(* CODESYS project ast_v1_0.library
   Company: Deprag
   Version: 1.0
   Placeholder: AST_V1_0
   Title: AST_V1_0

Project tree, tasks and I/O mapping:
  Data types/
    AST11/
      data type tAST11
      data type tAST11control
      data type tAST11data
      data type tAST11Rx
      data type tAST11state
      data type tAST11Tx
    AST40/
      data type tAST40
      data type tAST40control
      data type tAST40data
      data type tAST40Rx
      data type tAST40state
      data type tAST40Tx
    AST6/
      data type tAST6
      data type tAST6control
      data type tAST6data
      data type tAST6Rx
      data type tAST6state
      data type tAST6Tx
  Global Variables/
    global variables Globale_Variablen
  POUs/
    AST11/
      function block FB_AST11 [ST]: mthConvertControlSignal, mthConvertFinalData, mthConvertStatusSignal
      function FC_ConvertUnitAST11 [ST]
    AST40/
      function block FB_AST40 [ST]: mthConvertControlSignal, mthConvertFinalData, mthConvertStatusSignal
      function FC_ConvertUnitAST40 [ST]
    AST6/
      function block FB_AST6 [ST]: mthConvertControlSignal, mthConvertFinalData, mthConvertStatusSignal
      function FC_ConvertUnitAST6 [ST]
    Internal/
      function Merge_Byte2DInt [ST]
      function Merge_Byte2Int [ST]
      function Merge_Byte2Real [ST]
      function Split_Int2Byte [ST]
  Version/
    global variables Global_Version
  Visualizations/
*)

// Data types/AST11/tAST11
TYPE tAST11 :
	STRUCT
		Control			: tAST11control;
		State			: tAST11state;
		Data			: tAST11data;
	END_STRUCT
END_TYPE

// Data types/AST11/tAST11control
TYPE tAST11control :
	STRUCT
		Start			: BOOL := FALSE;
		Stop			: BOOL := FALSE;
		AutoStop		: BOOL := FALSE;
		Reload			: BOOL := FALSE;
		StartRelease	: BOOL := FALSE;
		ProgIn2			: BOOL := FALSE;
		FC_PartSensor	: BOOL := FALSE;
		FC_ReleasePart	: BOOL := FALSE;
		FC_ErrorReset	: BOOL := FALSE;
		DataSaved		: BOOL := FALSE;
		ResetPowerunit	: BOOL := FALSE;
		ResetMaintenance: BOOL := FALSE;
		ResetCycleStarted: BOOL := FALSE;
		Heartbeat		: BOOL := FALSE;
		ProgramNo		: INT := 0;
	END_STRUCT
END_TYPE

// Data types/AST11/tAST11data
TYPE tAST11data :
	STRUCT
		fdProg			: INT;
		fdStatus		: INT;
		fdTime			: REAL;

		fdStep1			: DINT;
		fdTorque1		: REAL;
		fdAngle1		: DINT;

		fdStep2			: DINT;
		fdTorque2		: REAL;
		fdAngle2		: DINT;

		fdStep3			: DINT;
		fdTorque3		: REAL;
		fdAngle3		: DINT;

		fdStepNOk		: DINT;
		fdTorqueNOk		: REAL;
		fdAngleNOk		: DINT;

		fdTorqueUnit	: INT;

		FC_Status		: INT;
		FC_TargetCount	: INT;
		FC_ActualCount	: INT;
	END_STRUCT
END_TYPE

// Data types/AST11/tAST11Rx
TYPE
	tAST11Rx : ARRAY[0..71] OF BYTE;
END_TYPE

// Data types/AST11/tAST11state
TYPE tAST11state :

	STRUCT
		SystemOK		: BOOL := FALSE;
		Ready			: BOOL := FALSE;
		OK				: BOOL := FALSE;
		NOK				: BOOL := FALSE;
		FC_PartActive	: BOOL := FALSE;
		FC_ChangePart	: BOOL := FALSE;
		ProgOut8		: BOOL := FALSE;
		DataAvailable	: BOOL := FALSE;

		ExtStop			: BOOL := FALSE;
		CycleActive		: BOOL := FALSE;
		CycleStarted	: BOOL := FALSE;
		Heartbeat		: BOOL := FALSE;

		SysStatus		: INT := 0;
	END_STRUCT
END_TYPE

// Data types/AST11/tAST11Tx
TYPE tAST11Tx : ARRAY[0..3] OF BYTE;
END_TYPE

// Data types/AST40/tAST40
TYPE tAST40 :
	STRUCT
		Control			: tAST40control;
		State			: tAST40state;
		Data			: tAST40data;
	END_STRUCT
END_TYPE

// Data types/AST40/tAST40control
TYPE tAST40control :
	STRUCT
		FCErrReset		: BOOL := FALSE;
		FCPartSensor	: BOOL := FALSE;
		FCReleasePart	: BOOL := FALSE;
		ReleaseStart	: BOOL := FALSE;
		Start			: BOOL := FALSE;
		Reload			: BOOL := FALSE;
		In1				: BOOL := FALSE;
		In2				: BOOL := FALSE;
		In3				: BOOL := FALSE;
		In4				: BOOL := FALSE;
		Res1			: BOOL := FALSE;
		Res2			: BOOL := FALSE;
		Res3			: BOOL := FALSE;
		Res4			: BOOL := FALSE;
		Res5			: BOOL := FALSE;
		Res6			: BOOL := FALSE;
		ProgramNo		: INT  := 0;
		In5				: BOOL := FALSE;
		In6				: BOOL := FALSE;
		In7				: BOOL := FALSE;
		In8				: BOOL := FALSE;
		In9				: BOOL := FALSE;
		In10			: BOOL := FALSE;
		In11			: BOOL := FALSE;
		In12			: BOOL := FALSE;
		UniInRes1		: BOOL := FALSE;
		UniInRes2		: BOOL := FALSE;
		UniInRes3		: BOOL := FALSE;
		UniInRes4		: BOOL := FALSE;
		UniInRes5		: BOOL := FALSE;
		UniInRes6		: BOOL := FALSE;
		UniInRes7		: BOOL := FALSE;
		UniInRes8		: BOOL := FALSE;
		DataSaved		: BOOL := FALSE;
		Heartbeat		: BOOL := FALSE;
		InRes1			: BOOL := FALSE;
		InRes2			: BOOL := FALSE;
		InRes3			: BOOL := FALSE;
		InRes4			: BOOL := FALSE;
		InRes5			: BOOL := FALSE;
		InRes6			: BOOL := FALSE;
		InRes7			: BOOL := FALSE;
		InRes8			: BOOL := FALSE;
		InRes9			: BOOL := FALSE;
		InRes10			: BOOL := FALSE;
		InRes11			: BOOL := FALSE;
		InRes12			: BOOL := FALSE;
		InRes13			: BOOL := FALSE;
		InRes14			: BOOL := FALSE;
	END_STRUCT
END_TYPE

// Data types/AST40/tAST40data
TYPE tAST40data :
	STRUCT
		fdProg			: INT;
		fdStatus		: INT;
		fdTime			: REAL;

		fdStep1			: DINT;
		fdMinTorque1	: REAL;
		fdTarTorque1	: REAL;
		fdMaxTorque1	: REAL;
		fdTorque1		: REAL;
		fdMinAngle1		: DINT;
		fdTarAngle1		: DINT;
		fdMaxAngle1		: DINT;
		fdAngle1		: REAL;

		fdStep2			: DINT;
		fdMinTorque2	: REAL;
		fdTarTorque2	: REAL;
		fdMaxTorque2	: REAL;
		fdTorque2		: REAL;
		fdMinAngle2		: DINT;
		fdTarAngle2		: DINT;
		fdMaxAngle2		: DINT;
		fdAngle2		: REAL;

		fdStep3			: DINT;
		fdMinTorque3	: REAL;
		fdTarTorque3	: REAL;
		fdMaxTorque3	: REAL;
		fdTorque3		: REAL;
		fdMinAngle3		: DINT;
		fdTarAngle3		: DINT;
		fdMaxAngle3		: DINT;
		fdAngle3		: REAL;

		fdStepNOk		: DINT;
		fdMinTorqueNOk	: REAL;
		fdTarTorqueNOk	: REAL;
		fdMaxTorqueNOk	: REAL;
		fdTorqueNOk		: REAL;
		fdMinAngleNOk	: DINT;
		fdTarAngleNOk	: DINT;
		fdMaxAngleNOk	: DINT;
		fdAngleNOk		: REAL;

		fdTorqueUnit	: INT;
	END_STRUCT
END_TYPE

// Data types/AST40/tAST40Rx
TYPE
	tAST40Rx : ARRAY[0..169] OF BYTE;
END_TYPE

// Data types/AST40/tAST40state
TYPE tAST40state :
	STRUCT
		SystemOK		: BOOL := FALSE;
		Ready			: BOOL := FALSE;
		OK				: BOOL := FALSE;
		NOK				: BOOL := FALSE;
		StatusHSres		: BOOL := FALSE;
		Sto1active		: BOOL := FALSE;
		Sto2active		: BOOL := FALSE;
		CycleActive		: BOOL := FALSE;
		ProgOut1		: BOOL := FALSE;
		ProgOut2		: BOOL := FALSE;
		ProgOut3		: BOOL := FALSE;
		ProgOut4		: BOOL := FALSE;
		FC_LockPart		: BOOL := FALSE;
		StatLTres		: BOOL := FALSE;
		FC_CycleDone	: BOOL := FALSE;
		Reload			: BOOL := FALSE;
		ProgOut5		: BOOL := FALSE;
		ProgOut6		: BOOL := FALSE;
		ProgOut7		: BOOL := FALSE;
		ProgOut8		: BOOL := FALSE;
		ProgOut9		: BOOL := FALSE;
		ProgOut10		: BOOL := FALSE;
		ProgOut11		: BOOL := FALSE;
		ProgOut12		: BOOL := FALSE;
		UniOutRes1		: BOOL := FALSE;
		UniOutRes2		: BOOL := FALSE;
		UniOutRes3		: BOOL := FALSE;
		UniOutRes4		: BOOL := FALSE;
		UniOutRes5		: BOOL := FALSE;
		UniOutRes6		: BOOL := FALSE;
		UniOutRes7		: BOOL := FALSE;
		UniOutRes8		: BOOL := FALSE;
		DataAvailable	: BOOL := FALSE;
		Heartbeat		: BOOL := FALSE;
		OutRes1			: BOOL := FALSE;
		OutRes2			: BOOL := FALSE;
		OutRes3			: BOOL := FALSE;
		OutRes4			: BOOL := FALSE;
		OutRes5			: BOOL := FALSE;
		OutRes6			: BOOL := FALSE;
		OutRes7			: BOOL := FALSE;
		OutRes8			: BOOL := FALSE;
		OutRes9			: BOOL := FALSE;
		OutRes10		: BOOL := FALSE;
		OutRes11		: BOOL := FALSE;
		OutRes12		: BOOL := FALSE;
		OutRes13		: BOOL := FALSE;
		OutRes14		: BOOL := FALSE;
		HW_FCErrReset	: BOOL := FALSE;
		HW_FCPartSensor	: BOOL := FALSE;
		HW_FCPartRelease: BOOL := FALSE;
		HW_ReleaseStart	: BOOL := FALSE;
		HW_Start		: BOOL := FALSE;
		HW_Reload		: BOOL := FALSE;
		HW_ProgIn1		: BOOL := FALSE;
		HW_ProgIn2		: BOOL := FALSE;
		HW_ProgIn3		: BOOL := FALSE;
		HW_ProgIn4		: BOOL := FALSE;
		HW_Res1			: BOOL := FALSE;
		HW_Res2			: BOOL := FALSE;
		HW_Res3			: BOOL := FALSE;
		HW_Res4			: BOOL := FALSE;
		HW_Res5			: BOOL := FALSE;
		HW_Res6			: BOOL := FALSE;
		AnalogStop		: INT  := 0;
		SysStatus		: INT  := 0;
	END_STRUCT
END_TYPE

// Data types/AST40/tAST40Tx
TYPE tAST40Tx : ARRAY[0..17] OF BYTE;
END_TYPE

// Data types/AST6/tAST6
TYPE tAST6 :
	STRUCT
		Control			: tAST6control;
		State			: tAST6state;
		Data			: tAST6data;
	END_STRUCT
END_TYPE

// Data types/AST6/tAST6control
TYPE tAST6control :
	STRUCT
		Start			: BOOL := FALSE;
		ProgIn1			: BOOL := FALSE;
		ProgIn2			: BOOL := FALSE;
		ProgIn3			: BOOL := FALSE;
		ProgIn4			: BOOL := FALSE;
		ProgIn5			: BOOL := FALSE;
		ProgIn6			: BOOL := FALSE;
		ProgramNo		: INT := 0;
		DataSaved		: BOOL := FALSE;
		Heartbeat		: BOOL := FALSE;
	END_STRUCT
END_TYPE

// Data types/AST6/tAST6data
TYPE tAST6data :
	STRUCT
		fdProg			: INT;
		fdStatus		: INT;
		fdTime			: REAL;

		fdStep1			: DINT;
		fdTorque1		: REAL;
		fdAngle1		: DINT;

		fdStep2			: DINT;
		fdTorque2		: REAL;
		fdAngle2		: DINT;

		fdStep3			: DINT;
		fdTorque3		: REAL;
		fdAngle3		: DINT;

		fdStepNOk		: DINT;
		fdTorqueNOk		: REAL;
		fdAngleNOk		: DINT;

		fdTorqueUnit	: INT;

	END_STRUCT
END_TYPE

// Data types/AST6/tAST6Rx
TYPE
	tAST6Rx : ARRAY[0..169] OF BYTE;
END_TYPE

// Data types/AST6/tAST6state
TYPE tAST6state :

	STRUCT
		SystemOK		: BOOL := FALSE;
		Ready			: BOOL := FALSE;
		OK				: BOOL := FALSE;
		NOK				: BOOL := FALSE;
		ProgOut1		: BOOL := FALSE;
		ProgOut2		: BOOL := FALSE;
		ProgOut3		: BOOL := FALSE;
		ProgOut4		: BOOL := FALSE;

		DataAvailable	: BOOL := FALSE;
		Heartbeat		: BOOL := FALSE;

		HW_Start		: BOOL := FALSE;
		HW_ProgIn1		: BOOL := FALSE;
		HW_ProgIn2		: BOOL := FALSE;
		HW_ProgIn3		: BOOL := FALSE;
		HW_ProgIn4		: BOOL := FALSE;
		HW_ProgIn5		: BOOL := FALSE;
		HW_ProgIn6		: BOOL := FALSE;

		SysStatus		: INT := 0;
	END_STRUCT
END_TYPE

// Data types/AST6/tAST6Tx
TYPE tAST6Tx : ARRAY[0..17] OF BYTE;
END_TYPE

// Global Variables/Globale_Variablen
{attribute 'Tc2GvlVarNames'}
VAR_GLOBAL
END_VAR

// Version/Global_Version
// This function has been automatically generated from the project information.
VAR_GLOBAL CONSTANT
	{attribute 'const_non_replaced'}
	{attribute 'linkalways'}
	stLibVersion_AST_V1_0 : ST_LibVersion := (iMajor := 1, iMinor := 0, iBuild := 0, iRevision := 0, sVersion := '1.0');
END_VAR

// POUs/AST11/FB_AST11
FUNCTION_BLOCK FB_AST11
VAR_INPUT
	RxAST11			: tAST11Rx;			(* output from HW AST11 *)
	Control			: tAST11control;
END_VAR
VAR_OUTPUT
	TxAST11			: tAST11Tx;			(* input for HW AST11 *)
	State			: tAST11State;
	Data			: tAST11data;
END_VAR
{library private}
VAR
	ArrTmpByte		: ARRAY[1..2] OF BYTE;
END_VAR

(* ------------------------------------------------------------------------------ *)
(*	AST11 - Control                                                                *)
(* ------------------------------------------------------------------------------ *)

		mthConvertStatusSignal();
		mthConvertFinalData();
		mthConvertControlSignal();

ACTION mthConvertControlSignal:

	TxAST11[0].0	:= Control.Start;
	TxAST11[0].1	:= (NOT Control.Start AND Control.AutoStop) OR Control.Stop;
	TxAST11[0].2	:= Control.Reload;
	TxAST11[0].3	:= Control.StartRelease;
	TxAST11[0].4	:= FALSE;
	TxAST11[0].5	:= Control.FC_PartSensor;
	TxAST11[0].6	:= Control.FC_ErrorReset;
	TxAST11[0].7	:= Control.FC_ReleasePart;

	TxAST11[1].0	:= Control.ProgIn2;
	TxAST11[1].1	:= Control.DataSaved;
	TxAST11[1].2	:= Control.ResetPowerunit;
	TxAST11[1].3	:= Control.Heartbeat := State.Heartbeat;
	TxAST11[1].4	:= Control.ResetMaintenance;
	TxAST11[1].5	:= Control.ResetCycleStarted;
	TxAST11[1].6	:= FALSE;
	TxAST11[1].7	:= FALSE;

	ArrTmpByte	:= Split_Int2Byte(Control.ProgramNo);
	TxAST11[2]	:= ArrTmpByte[1];
	TxAST11[3]	:= ArrTmpByte[2];
END_ACTION

ACTION mthConvertFinalData:
(* General Data *)
	Data.fdProg				:= Merge_Byte2Int(
											RxAST11[8],
											RxAST11[9]);
	Data.fdStatus			:= Merge_Byte2Int(
											RxAST11[10],
											RxAST11[11]);
	Data.fdTime				:= Merge_Byte2Real(
											RxAST11[12],
											RxAST11[13],
											RxAST11[14],
											RxAST11[15]);
(* Data Step 1 *)
	Data.fdStep1			:= Merge_Byte2DInt(
											RxAST11[16],
											RxAST11[17],
											RxAST11[18],
											RxAST11[19]);
	Data.fdTorque1			:= Merge_Byte2Real(
											RxAST11[20],
											RxAST11[21],
											RxAST11[22],
											RxAST11[23]);
	Data.fdAngle1			:= Merge_Byte2DInt(
											RxAST11[24],
											RxAST11[25],
											RxAST11[26],
											RxAST11[27]);
(* Data Step 2 *)
	Data.fdStep2			:= Merge_Byte2DInt(
											RxAST11[28],
											RxAST11[29],
											RxAST11[30],
											RxAST11[31]);
	Data.fdTorque2			:= Merge_Byte2Real(
											RxAST11[32],
											RxAST11[33],
											RxAST11[34],
											RxAST11[35]);
	Data.fdAngle2			:= Merge_Byte2DInt(
											RxAST11[36],
											RxAST11[37],
											RxAST11[38],
											RxAST11[39]);
(* Data Step 3 *)
	Data.fdStep3			:= Merge_Byte2DInt(
											RxAST11[40],
											RxAST11[41],
											RxAST11[42],
											RxAST11[43]);
	Data.fdTorque3			:= Merge_Byte2Real(
											RxAST11[44],
											RxAST11[45],
											RxAST11[46],
											RxAST11[47]);
	Data.fdAngle3			:= Merge_Byte2DInt(
											RxAST11[48],
											RxAST11[49],
											RxAST11[50],
											RxAST11[51]);
(* Data Step NOK *)
	Data.fdStepNOk			:= Merge_Byte2DInt(
											RxAST11[52],
											RxAST11[53],
											RxAST11[54],
											RxAST11[55]);
	Data.fdTorqueNOk		:= Merge_Byte2Real(
											RxAST11[56],
											RxAST11[57],
											RxAST11[58],
											RxAST11[59]);
	Data.fdAngleNOk			:= Merge_Byte2DInt(
											RxAST11[60],
											RxAST11[61],
											RxAST11[62],
											RxAST11[63]);
(* Data Torque Unit *)
	Data.fdTorqueUnit		:= Merge_Byte2Int(
											RxAST11[64],
											RxAST11[65]);


(* Data F-Control *)
	Data.FC_Status			:= Merge_Byte2Int(
											RxAST11[66],
											RxAST11[67]);

	Data.FC_TargetCount		:= Merge_Byte2Int(
											RxAST11[68],
											RxAST11[69]);

	Data.FC_ActualCount		:= Merge_Byte2Int(
											RxAST11[70],
											RxAST11[71]);
END_ACTION

ACTION mthConvertStatusSignal:

	State.SystemOK			:= RxAST11[4].0;
	State.Ready				:= RxAST11[4].1;
	State.OK				:= RxAST11[4].2;
	State.NOK				:= RxAST11[4].3;
	State.FC_ChangePart		:= RxAST11[4].4;
	State.FC_PartActive		:= RxAST11[4].5;
	State.ProgOut8			:= RxAST11[4].6;
	State.Heartbeat			:= RxAST11[4].7;

	State.DataAvailable		:= RxAST11[5].0;
	State.ExtStop			:= RxAST11[5].1;
	State.CycleActive		:= RxAST11[5].2;
	State.CycleStarted		:= RxAST11[5].3;

	State.SysStatus			:= Merge_Byte2Int(
									RxAST11[6],
									RxAST11[7]);
END_ACTION

END_FUNCTION_BLOCK

// POUs/Internal/Split_Int2Byte
FUNCTION Split_Int2Byte : ARRAY[1..2] OF BYTE
{library private}
VAR_INPUT
	I		: INT;
END_VAR
VAR
	pt		: POINTER TO ARRAY[1..2] OF BYTE;
END_VAR

pt		:=	ADR(I);

Split_Int2Byte := pt^;

END_FUNCTION

// POUs/Internal/Merge_Byte2Int
FUNCTION Merge_Byte2Int : INT
{library private}
VAR_INPUT
	B0		: BYTE;
	B1		: BYTE;
END_VAR
VAR
	TmpVar	: WORD;
	pt		: POINTER TO INT;
END_VAR

TmpVar	:=	SHL(BYTE_TO_WORD(B1),8) OR BYTE_TO_WORD(B0);
pt		:=	ADR(TmpVar);

Merge_Byte2Int := pt^;

END_FUNCTION

// POUs/Internal/Merge_Byte2Real
FUNCTION Merge_Byte2Real : REAL
{library private}
VAR_INPUT
	B0		: BYTE;
	B1		: BYTE;
	B2		: BYTE;
	B3		: BYTE;
END_VAR
VAR
	TmpVar	: DWORD;
	pt		: POINTER TO REAL;
END_VAR

TmpVar	:=	SHL(SHL(SHL(BYTE_TO_DWORD(B3),8) OR BYTE_TO_DWORD(B2),8) OR BYTE_TO_DWORD(B1),8) OR BYTE_TO_DWORD(B0);
pt		:=	ADR(TmpVar);

Merge_Byte2Real := pt^;

END_FUNCTION

// POUs/Internal/Merge_Byte2DInt
FUNCTION Merge_Byte2DInt : DINT
{library private}
VAR_INPUT
	B0		: BYTE;
	B1		: BYTE;
	B2		: BYTE;
	B3		: BYTE;
END_VAR
VAR
	TmpVar	: DWORD;
	pt		: POINTER TO DINT;
END_VAR

TmpVar	:=	SHL(SHL(SHL(BYTE_TO_DWORD(B3),8) OR BYTE_TO_DWORD(B2),8) OR BYTE_TO_DWORD(B1),8) OR BYTE_TO_DWORD(B0);
pt		:=	ADR(TmpVar);

Merge_Byte2DInt := pt^;

END_FUNCTION

// POUs/AST11/FC_ConvertUnitAST11
FUNCTION FC_ConvertUnitAST11 : STRING[5]
(*
	0 = "Nm"
	1 = "Ncm"
	2 = "ft-lb"
	3 = "in-lb"
	4 = "kg-m"
	5 = "kg-cm"
*)
VAR_INPUT
	TorqueUnit	: INT;
END_VAR
{library private}
VAR
END_VAR

CASE TorqueUnit OF
	0:	FC_ConvertUnitAST11	:= 'Nm';
	1:	FC_ConvertUnitAST11	:= 'Ncm';
	2:	FC_ConvertUnitAST11	:= 'ft-lb';
	3:	FC_ConvertUnitAST11	:= 'in-lb';
	4:	FC_ConvertUnitAST11	:= 'kg-m';
	5:	FC_ConvertUnitAST11	:= 'kg-cm';
ELSE
	FC_ConvertUnitAST11 := '';
END_CASE

END_FUNCTION

// POUs/AST40/FB_AST40
FUNCTION_BLOCK FB_AST40
VAR_INPUT
	RxAST40			: tAST40Rx;			(* output from HW AST40 *)
	Control			: tAST40control;
END_VAR

VAR_OUTPUT
	TxAST40			: tAST40Tx;			(* input for HW AST40 *)
	State			: tAST40State;
	Data			: tAST40data;
END_VAR
{library private}
VAR
	ArrTmpByte		: ARRAY[1..2] OF BYTE;
END_VAR

(* ------------------------------------------------------------------------------ *)
(*	AST40 - Control                                                                *)
(* ------------------------------------------------------------------------------ *)

		mthConvertStatusSignal();
		mthConvertFinalData();
		mthConvertControlSignal();

ACTION mthConvertControlSignal:
	TxAST40[0].0	:= Control.FCErrReset;
	TxAST40[0].1	:= Control.FCPartSensor;
	TxAST40[0].2	:= Control.FCReleasePart;
	TxAST40[0].3	:= Control.ReleaseStart;
	TxAST40[0].4	:= Control.Start;
	TxAST40[0].5	:= Control.Reload;
	TxAST40[0].6	:= Control.In1;
	TxAST40[0].7	:= Control.In2;

	TxAST40[1].0	:= Control.In3;
	TxAST40[1].1	:= Control.In4;
	TxAST40[1].2	:= Control.Res1;
	TxAST40[1].3	:= Control.Res2;
	TxAST40[1].4	:= Control.Res3;
	TxAST40[1].5	:= Control.Res4;
	TxAST40[1].6	:= Control.Res5;
	TxAST40[1].7	:= Control.Res6;

	ArrTmpByte		:= Split_Int2Byte(Control.ProgramNo);
	TxAST40[2]		:= ArrTmpByte[1];
	TxAST40[3]		:= ArrTmpByte[2];

	TxAST40[4].0	:= Control.In5;
	TxAST40[4].1	:= Control.In6;
	TxAST40[4].2	:= Control.In7;
	TxAST40[4].3	:= Control.In8;
	TxAST40[4].4	:= Control.In9;
	TxAST40[4].5	:= Control.In10;
	TxAST40[4].6	:= Control.In11;
	TxAST40[4].7	:= Control.In12;

	TxAST40[5].0	:= Control.UniInRes1;
	TxAST40[5].1	:= Control.UniInRes2;
	TxAST40[5].2	:= Control.UniInRes3;
	TxAST40[5].3	:= Control.UniInRes4;
	TxAST40[5].4	:= Control.UniInRes5;
	TxAST40[5].5	:= Control.UniInRes6;
	TxAST40[5].6	:= Control.UniInRes7;
	TxAST40[5].7	:= Control.UniInRes8;

	TxAST40[6].0	:= Control.DataSaved;
	TxAST40[6].1	:= Control.Heartbeat := State.Heartbeat;
	TxAST40[6].2	:= Control.InRes1;
	TxAST40[6].3	:= Control.InRes2;
	TxAST40[6].4	:= Control.InRes3;
	TxAST40[6].5	:= Control.InRes4;
	TxAST40[6].6	:= Control.InRes5;
	TxAST40[6].7	:= Control.InRes6;

	TxAST40[7].0	:= Control.InRes7;
	TxAST40[7].1	:= Control.InRes8;
	TxAST40[7].2	:= Control.InRes9;
	TxAST40[7].3	:= Control.InRes10;
	TxAST40[7].4	:= Control.InRes11;
	TxAST40[7].5	:= Control.InRes12;
	TxAST40[7].6	:= Control.InRes13;
	TxAST40[7].7	:= Control.InRes14;

	ArrTmpByte		:= Split_Int2Byte(1);
	TxAST40[8]		:= ArrTmpByte[1];
	TxAST40[9]		:= ArrTmpByte[2];
END_ACTION

ACTION mthConvertFinalData:
(* General Data *)
	Data.fdProg			:= Merge_Byte2Int(
								RxAST40[16],
								RxAST40[17]);
	Data.fdStatus		:= Merge_Byte2Int(
								RxAST40[18],
								RxAST40[19]);
	Data.fdTime			:= Merge_Byte2Real(
								RxAST40[20],
								RxAST40[21],
								RxAST40[22],
								RxAST40[23]);
(* Data Step 1 *)
	Data.fdStep1		:= Merge_Byte2DInt(
								RxAST40[24],
								RxAST40[25],
								RxAST40[26],
								RxAST40[27]);
	Data.fdMinTorque1	:= Merge_Byte2Real(
								RxAST40[28],
								RxAST40[29],
								RxAST40[30],
								RxAST40[31]);
	Data.fdTarTorque1	:= Merge_Byte2Real(
								RxAST40[32],
								RxAST40[33],
								RxAST40[34],
								RxAST40[35]);
	Data.fdMaxTorque1	:= Merge_Byte2Real(
								RxAST40[36],
								RxAST40[37],
								RxAST40[38],
								RxAST40[39]);
	Data.fdTorque1		:= Merge_Byte2Real(
								RxAST40[40],
								RxAST40[41],
								RxAST40[42],
								RxAST40[43]);
	Data.fdMinAngle1	:= Merge_Byte2DInt(
								RxAST40[44],
								RxAST40[45],
								RxAST40[46],
								RxAST40[47]);
	Data.fdTarAngle1	:= Merge_Byte2DInt(
								RxAST40[48],
								RxAST40[49],
								RxAST40[50],
								RxAST40[51]);
	Data.fdMaxAngle1	:= Merge_Byte2DInt(
								RxAST40[52],
								RxAST40[53],
								RxAST40[54],
								RxAST40[55]);
	Data.fdAngle1		:= Merge_Byte2Real(
								RxAST40[56],
								RxAST40[57],
								RxAST40[58],
								RxAST40[59]);
(* Data Step 2 *)
	Data.fdStep2		:= Merge_Byte2DInt(
								RxAST40[60],
								RxAST40[61],
								RxAST40[62],
								RxAST40[63]);
	Data.fdMinTorque2	:= Merge_Byte2Real(
								RxAST40[64],
								RxAST40[65],
								RxAST40[66],
								RxAST40[67]);
	Data.fdTarTorque2	:= Merge_Byte2Real(
								RxAST40[68],
								RxAST40[69],
								RxAST40[70],
								RxAST40[71]);
	Data.fdMaxTorque2	:= Merge_Byte2Real(
								RxAST40[72],
								RxAST40[73],
								RxAST40[74],
								RxAST40[75]);
	Data.fdTorque2		:= Merge_Byte2Real(
								RxAST40[76],
								RxAST40[77],
								RxAST40[78],
								RxAST40[79]);
	Data.fdMinAngle2	:= Merge_Byte2DInt(
								RxAST40[80],
								RxAST40[81],
								RxAST40[82],
								RxAST40[83]);
	Data.fdTarAngle2	:= Merge_Byte2DInt(
								RxAST40[84],
								RxAST40[85],
								RxAST40[86],
								RxAST40[87]);
	Data.fdMaxAngle2	:= Merge_Byte2DInt(
								RxAST40[88],
								RxAST40[89],
								RxAST40[90],
								RxAST40[91]);
	Data.fdAngle2		:= Merge_Byte2Real(
								RxAST40[92],
								RxAST40[93],
								RxAST40[94],
								RxAST40[95]);
(* Data Step 3 *)
	Data.fdStep3		:= Merge_Byte2DInt(
								RxAST40[96],
								RxAST40[97],
								RxAST40[98],
								RxAST40[99]);
	Data.fdMinTorque3	:= Merge_Byte2Real(
								RxAST40[100],
								RxAST40[101],
								RxAST40[102],
								RxAST40[103]);
	Data.fdTarTorque3	:= Merge_Byte2Real(
								RxAST40[104],
								RxAST40[105],
								RxAST40[106],
								RxAST40[107]);
	Data.fdMaxTorque3	:= Merge_Byte2Real(
								RxAST40[108],
								RxAST40[109],
								RxAST40[110],
								RxAST40[111]);
	Data.fdTorque3		:= Merge_Byte2Real(
								RxAST40[112],
								RxAST40[113],
								RxAST40[114],
								RxAST40[115]);
	Data.fdMinAngle3	:= Merge_Byte2DInt(
								RxAST40[116],
								RxAST40[117],
								RxAST40[118],
								RxAST40[119]);
	Data.fdTarAngle3	:= Merge_Byte2DInt(
								RxAST40[120],
								RxAST40[121],
								RxAST40[122],
								RxAST40[123]);
	Data.fdMaxAngle3	:= Merge_Byte2DInt(
								RxAST40[124],
								RxAST40[125],
								RxAST40[126],
								RxAST40[127]);
	Data.fdAngle3		:= Merge_Byte2Real(
								RxAST40[128],
								RxAST40[129],
								RxAST40[130],
								RxAST40[131]);
(* Data Step NOK *)
	Data.fdStepNOk		:= Merge_Byte2DInt(
								RxAST40[132],
								RxAST40[133],
								RxAST40[134],
								RxAST40[135]);
	Data.fdMinTorqueNOk	:= Merge_Byte2Real(
								RxAST40[136],
								RxAST40[137],
								RxAST40[138],
								RxAST40[139]);
	Data.fdTarTorqueNOk	:= Merge_Byte2Real(
								RxAST40[140],
								RxAST40[141],
								RxAST40[142],
								RxAST40[143]);
	Data.fdMaxTorqueNOk	:= Merge_Byte2Real(
								RxAST40[144],
								RxAST40[145],
								RxAST40[146],
								RxAST40[147]);
	Data.fdTorqueNOk	:= Merge_Byte2Real(
								RxAST40[148],
								RxAST40[149],
								RxAST40[150],
								RxAST40[151]);
	Data.fdMinAngleNOk	:= Merge_Byte2DInt(
								RxAST40[152],
								RxAST40[153],
								RxAST40[154],
								RxAST40[155]);
	Data.fdTarAngleNOk	:= Merge_Byte2DInt(
								RxAST40[156],
								RxAST40[157],
								RxAST40[158],
								RxAST40[159]);
	Data.fdMaxAngleNOk	:= Merge_Byte2DInt(
								RxAST40[160],
								RxAST40[161],
								RxAST40[162],
								RxAST40[163]);
	Data.fdAngleNOk		:= Merge_Byte2Real(
								RxAST40[164],
								RxAST40[165],
								RxAST40[166],
								RxAST40[167]);
(* Data Torque Unit *)
	Data.fdTorqueUnit	:= Merge_Byte2Int(
								RxAST40[168],
								RxAST40[169]);
END_ACTION

ACTION mthConvertStatusSignal:
	State.SystemOK			:= RxAST40[4].0;
	State.Ready				:= RxAST40[4].1;
	State.OK				:= RxAST40[4].2;
	State.NOK				:= RxAST40[4].3;
	State.StatusHSres		:= RxAST40[4].4;
	State.Sto1active		:= RxAST40[4].5;
	State.Sto2active		:= RxAST40[4].6;
	State.CycleActive		:= RxAST40[4].7;
	State.ProgOut1			:= RxAST40[5].0;
	State.ProgOut2			:= RxAST40[5].1;
	State.ProgOut3			:= RxAST40[5].2;
	State.ProgOut4			:= RxAST40[5].3;
	State.FC_LockPart		:= RxAST40[5].4;
	State.StatLTres			:= RxAST40[5].5;
	State.FC_CycleDone		:= RxAST40[5].6;
	State.Reload			:= RxAST40[5].7;

	State.ProgOut5			:= RxAST40[6].0;
	State.ProgOut6			:= RxAST40[6].1;
	State.ProgOut7			:= RxAST40[6].2;
	State.ProgOut8			:= RxAST40[6].3;
	State.ProgOut9			:= RxAST40[6].4;
	State.ProgOut10			:= RxAST40[6].5;
	State.ProgOut11			:= RxAST40[6].6;
	State.ProgOut12			:= RxAST40[6].7;
	State.UniOutRes1		:= RxAST40[7].0;
	State.UniOutRes2		:= RxAST40[7].1;
	State.UniOutRes3		:= RxAST40[7].2;
	State.UniOutRes4		:= RxAST40[7].3;
	State.UniOutRes5		:= RxAST40[7].4;
	State.UniOutRes6		:= RxAST40[7].5;
	State.UniOutRes7		:= RxAST40[7].6;
	State.UniOutRes8		:= RxAST40[7].7;

	State.DataAvailable		:= RxAST40[8].0;
	State.Heartbeat			:= RxAST40[8].1;
	State.OutRes1			:= RxAST40[8].2;
	State.OutRes2			:= RxAST40[8].3;
	State.OutRes3			:= RxAST40[8].4;
	State.OutRes4			:= RxAST40[8].5;
	State.OutRes5			:= RxAST40[8].6;
	State.OutRes6			:= RxAST40[8].7;
	State.OutRes7			:= RxAST40[9].0;
	State.OutRes8			:= RxAST40[9].1;
	State.OutRes9			:= RxAST40[9].2;
	State.OutRes10			:= RxAST40[9].3;
	State.OutRes11			:= RxAST40[9].4;
	State.OutRes12			:= RxAST40[9].5;
	State.OutRes13			:= RxAST40[9].6;
	State.OutRes14			:= RxAST40[9].7;

	State.HW_FCErrReset		:= RxAST40[10].0;
	State.HW_FCPartSensor	:= RxAST40[10].1;
	State.HW_FCPartRelease	:= RxAST40[10].2;
	State.HW_ReleaseStart	:= RxAST40[10].3;
	State.HW_Start			:= RxAST40[10].4;
	State.HW_Reload			:= RxAST40[10].5;
	State.HW_ProgIn1		:= RxAST40[10].6;
	State.HW_ProgIn2		:= RxAST40[10].7;
	State.HW_ProgIn3		:= RxAST40[11].0;
	State.HW_ProgIn4		:= RxAST40[11].1;
	State.HW_Res1			:= RxAST40[11].2;
	State.HW_Res2			:= RxAST40[11].3;
	State.HW_Res3			:= RxAST40[11].4;
	State.HW_Res4			:= RxAST40[11].5;
	State.HW_Res5			:= RxAST40[11].6;
	State.HW_Res6			:= RxAST40[11].7;


	State.AnalogStop		:= Merge_Byte2Int(
									RxAST40[12],
									RxAST40[13]);

	State.SysStatus			:= Merge_Byte2Int(
									RxAST40[14],
									RxAST40[15]);
END_ACTION

END_FUNCTION_BLOCK

// POUs/AST40/FC_ConvertUnitAST40
FUNCTION FC_ConvertUnitAST40 : STRING[5]
(*
	0 = "Nm"
	1 = "Ncm"
	2 = "ft-lb"
	3 = "in-lb"
	4 = "kg-m"
	5 = "kg-cm"
*)
VAR_INPUT
	TorqueUnit	: INT;
END_VAR
{library private}
VAR
END_VAR

CASE TorqueUnit OF
	0:	FC_ConvertUnitAST40	:= 'Nm';
	1:	FC_ConvertUnitAST40	:= 'Ncm';
	2:	FC_ConvertUnitAST40	:= 'ft-lb';
	3:	FC_ConvertUnitAST40	:= 'in-lb';
	4:	FC_ConvertUnitAST40	:= 'kg-m';
	5:	FC_ConvertUnitAST40	:= 'kg-cm';
ELSE
	FC_ConvertUnitAST40 := '';
END_CASE

END_FUNCTION

// POUs/AST6/FB_AST6
FUNCTION_BLOCK FB_AST6
VAR_INPUT
	RxAST6			: tAST6Rx;			(* output from HW AST6 *)
	Control			: tAST6control;
END_VAR
VAR_OUTPUT
	TxAST6			: tAST6Tx;			(* input for HW AST6 *)
	State			: tAST6State;
	Data			: tAST6data;
END_VAR
{library private}
VAR
	ArrTmpByte		: ARRAY[1..2] OF BYTE;
END_VAR

(* ------------------------------------------------------------------------------ *)
(*	AST6 - Control                                                                *)
(* ------------------------------------------------------------------------------ *)

		mthConvertStatusSignal();
		mthConvertFinalData();
		mthConvertControlSignal();

ACTION mthConvertControlSignal:
	TxAST6[0].0	:= FALSE;
	TxAST6[0].1	:= FALSE;
	TxAST6[0].2	:= FALSE;
	TxAST6[0].3	:= Control.ProgIn1;
	TxAST6[0].4	:= Control.Start;
	TxAST6[0].5	:= FALSE;
	TxAST6[0].6	:= Control.ProgIn3;
	TxAST6[0].7	:= Control.ProgIn4;

	TxAST6[1].0	:= Control.ProgIn5;
	TxAST6[1].1	:= Control.ProgIn6;
	TxAST6[1].2	:= Control.ProgIn2;
	TxAST6[1].3	:= FALSE;
	TxAST6[1].4	:= FALSE;
	TxAST6[1].5	:= FALSE;
	TxAST6[1].6	:= FALSE;
	TxAST6[1].7	:= FALSE;

(*	MEMCPY(destAddr:=ADR(TxAST6[2]) , srcAddr:= ADR(Control.ProgNo), n:= SIZEOF(Control.ProgNo));
*)
	ArrTmpByte	:= Split_Int2Byte(Control.ProgramNo);
	TxAST6[2]	:= ArrTmpByte[1];
	TxAST6[3]	:= ArrTmpByte[2];

	TxAST6[6].0	:= Control.DataSaved;
	TxAST6[6].1	:= Control.Heartbeat := State.Heartbeat;
	TxAST6[6].2	:= FALSE;
	TxAST6[6].3	:= FALSE;
	TxAST6[6].4	:= FALSE;
	TxAST6[6].5	:= FALSE;
	TxAST6[6].6	:= FALSE;
	TxAST6[6].7	:= FALSE;

	TxAST6[7].0	:= FALSE;
	TxAST6[7].1	:= FALSE;
	TxAST6[7].2	:= FALSE;
	TxAST6[7].3	:= FALSE;
	TxAST6[7].4	:= FALSE;
	TxAST6[7].5	:= FALSE;
	TxAST6[7].6	:= FALSE;
	TxAST6[7].7	:= FALSE;
END_ACTION

ACTION mthConvertFinalData:
(* General Data *)
	Data.fdProg			:= Merge_Byte2Int(
											RxAST6[16],
											RxAST6[17]);
	Data.fdStatus		:= Merge_Byte2Int(
											RxAST6[18],
											RxAST6[19]);
	Data.fdTime			:= Merge_Byte2Real(
											RxAST6[20],
											RxAST6[21],
											RxAST6[22],
											RxAST6[23]);
(* Data Step 1 *)
	Data.fdStep1			:= Merge_Byte2DInt(
											RxAST6[24],
											RxAST6[25],
											RxAST6[26],
											RxAST6[27]);
	Data.fdTorque1			:= Merge_Byte2Real(
											RxAST6[28],
											RxAST6[29],
											RxAST6[30],
											RxAST6[31]);
	Data.fdAngle1			:= Merge_Byte2DInt(
											RxAST6[32],
											RxAST6[33],
											RxAST6[34],
											RxAST6[35]);
(* Data Step 2 *)
	Data.fdStep2			:= Merge_Byte2DInt(
											RxAST6[36],
											RxAST6[37],
											RxAST6[38],
											RxAST6[39]);
	Data.fdTorque2			:= Merge_Byte2Real(
											RxAST6[40],
											RxAST6[41],
											RxAST6[42],
											RxAST6[43]);
	Data.fdAngle2			:= Merge_Byte2DInt(
											RxAST6[44],
											RxAST6[45],
											RxAST6[46],
											RxAST6[47]);
(* Data Step 3 *)
	Data.fdStep3			:= Merge_Byte2DInt(
											RxAST6[48],
											RxAST6[49],
											RxAST6[50],
											RxAST6[51]);
	Data.fdTorque3			:= Merge_Byte2Real(
											RxAST6[52],
											RxAST6[53],
											RxAST6[54],
											RxAST6[55]);
	Data.fdAngle3			:= Merge_Byte2DInt(
											RxAST6[56],
											RxAST6[57],
											RxAST6[58],
											RxAST6[59]);
(* Data Step NOK *)
	Data.fdStepNOk			:= Merge_Byte2DInt(
											RxAST6[60],
											RxAST6[61],
											RxAST6[62],
											RxAST6[63]);
	Data.fdTorqueNOk		:= Merge_Byte2Real(
											RxAST6[64],
											RxAST6[65],
											RxAST6[66],
											RxAST6[67]);
	Data.fdAngleNOk			:= Merge_Byte2DInt(
											RxAST6[68],
											RxAST6[69],
											RxAST6[70],
											RxAST6[71]);
(* Data Torque Unit *)
	Data.fdTorqueUnit		:= Merge_Byte2Int(
											RxAST6[72],
											RxAST6[73]);
END_ACTION

ACTION mthConvertStatusSignal:
	State.SystemOK			:= RxAST6[4].0;
	State.Ready				:= RxAST6[4].1;
	State.OK				:= RxAST6[4].2;
	State.NOK				:= RxAST6[4].3;

	State.DataAvailable		:= RxAST6[8].0;
	State.Heartbeat			:= RxAST6[8].1;

	State.HW_ProgIn1		:= RxAST6[10].3;
	State.HW_Start			:= RxAST6[10].4;
	State.HW_ProgIn3		:= RxAST6[10].6;
	State.HW_ProgIn4		:= RxAST6[10].7;
	State.HW_ProgIn5		:= RxAST6[11].0;
	State.HW_ProgIn6		:= RxAST6[11].1;
	State.HW_ProgIn2		:= RxAST6[11].2;

	State.SysStatus			:= Merge_Byte2Int(
									RxAST6[14],
									RxAST6[15]);
END_ACTION

END_FUNCTION_BLOCK

// POUs/AST6/FC_ConvertUnitAST6
FUNCTION FC_ConvertUnitAST6 : STRING[5]
(*
	0 = "Nm"
	1 = "Ncm"
	2 = "ft-lb"
	3 = "in-lb"
	4 = "kg-m"
	5 = "kg-cm"
*)
VAR_INPUT
	TorqueUnit	: INT;
END_VAR
{library private}
VAR
END_VAR

CASE TorqueUnit OF
	0:	FC_ConvertUnitAST6	:= 'Nm';
	1:	FC_ConvertUnitAST6	:= 'Ncm';
	2:	FC_ConvertUnitAST6	:= 'ft-lb';
	3:	FC_ConvertUnitAST6	:= 'in-lb';
	4:	FC_ConvertUnitAST6	:= 'kg-m';
	5:	FC_ConvertUnitAST6	:= 'kg-cm';
ELSE
	FC_ConvertUnitAST6 := '';
END_CASE;

END_FUNCTION
